(* CoDeSys 2.3.9.47 project: ATS_P6.pro *)
(* Libraries: STANDARD.LIB 5.6.98 12:03:02 *)

(* Task configuration *)
TASK Standard (PRIORITY := 0, INTERVAL := T#10ms);
	MAIN
END_TASK

(* POU MAIN, ST *)
PROGRAM MAIN
VAR
	sin_out : REAL; 	(*Output Signal*)
	sqr_out : REAL; 	(*Output Signal*)
	pwm_out	: REAL;		(*Output Signal*)
	t		: REAL:= 0; (*Input Signal*)
END_VAR
(*Sine Function Call*)
sin_out := SinusFunction(t);

(*Square Function Call*)
sqr_out	:= SquareSignal(t,2, 4);

(*PWM Function Call*)
pwm_out := PWMSignal(t, 10, 5);

(*Increment Time-Variable*)
t := t + 0.01;
END_PROGRAM

(* POU SinusFunction, ST *)
FUNCTION SinusFunction : REAL
VAR_INPUT
	t	:	REAL;		(*Input Time*)
END_VAR
VAR
	w	:	REAL := 1; 	(*Frequency*)
	A	:	REAL := 1;	(*Amplitude*)
	offs:	REAL := 0;	(*Offset*)
END_VAR
(*Generate Sine-Wave*)
SinusFunction := A*SIN(w*t) + offs;
END_FUNCTION

(* POU SquareSignal, ST *)
FUNCTION SquareSignal : REAL
VAR_INPUT
	t	:	REAL;		(*Input Time*)
	mini:	REAL;		(*Minimum Value*)
	maxi:	REAL;		(*Maximum Value*)
END_VAR
VAR
	w		:	REAL := 1; 	(*Frequency*)
	offs	:	REAL := 0;	(*Offset*)
	curr_sin:	REAL ;		(*Current Sine Wave*)
END_VAR
(*Generate Square-Wave*)

curr_sin := SIN(w*t);

IF curr_sin > 0 THEN
	SquareSignal := maxi + offs;
ELSE
	SquareSignal := mini + offs;
END_IF
END_FUNCTION

(* POU PWMSignal, ST *)
FUNCTION PWMSignal : REAL
VAR_INPUT
	t	:	REAL;		(*Input Time*)
	dc	:	REAL;		(*Input Duty Cicle*)
	per	:	REAL;		(*Input Period*)
END_VAR
VAR
	pi		:	REAL := 3.14159;
	w		:	REAL ;	(*Frequency*)
	th		:	REAL ;
	curr_sin:	REAL ;	(*Current Sine Wave*)
END_VAR
(*Generate PWM*)

(*Calculate Frequency using Period*)
w := (2*pi)/(per);
(*Generate Reference Wave*)
curr_sin := 0.5*SIN(w*t)+0.5;
(*Calculate Threshold*)
th := 1-((dc)/(100));
(*Check validity of Input Duty Call*)
IF (dc <= 0) OR (dc > 100) THEN
	PWMSignal := 0;
ELSE
(*Compare Reference Wave to Threshold*)
IF curr_sin > th THEN
	PWMSignal := 1;
ELSE
	PWMSignal := 0;
END_IF
END_IF
END_FUNCTION
